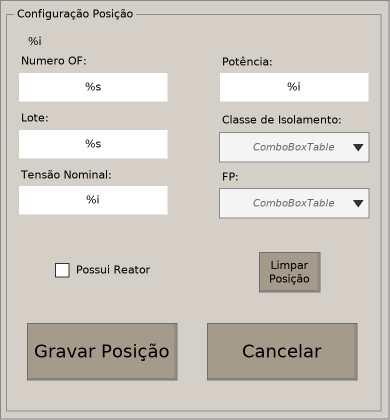
VISUALIZATION ConfigPosicao_2  // 390x420
VAR_IN_OUT
	bReator: BOOL;
	iOFnumber: INT;
	iSrlNumber: INT;
	
	
	
END_VAR
    GroupBox (6,6 375x405), "Configuração Posição"
        Checkbox (47,251 110x26), "Possui Reator", variable: gravarConfigPosicao020.bReator[1]
        Button (21,317 150x57), "Gravar Posição"
            OnMouseClick: CloseDialog Dialog=ConfigPosicao_2, Result=OK, NumpadKeypadSet=True
            OnMouseClick: execute { gravarConfigPosicao020(); }
        Button (201,317 150x57), "Cancelar"
            OnMouseClick: CloseDialog Dialog=ConfigPosicao_2, Result=Cancel, NumpadKeypadSet=True
        Button (253,246 61x40), "Limpar Posição"
            OnMouseClick: CloseDialog Dialog=ConfigPosicao_2, Result=Cancel, NumpadKeypadSet=True
            OnMouseClick: execute {
                gvl_p.aPositionsE020[gvl.actPos].numOF:='0';
                gvl_p.aPositionsE020[gvl.actPos].lote:='0';
                gvl_p.aPositionsE020[gvl.actPos].class:=0;
                gvl_p.aPositionsE020[gvl.actPos].pot:=0;
                gvl_p.aPositionsE020[gvl.actPos].cor:=0;
                IF gvl.totalPos[gvl.actEst] <> 0 THEN
                gvl.totalPos[gvl.actEst]:= gvl.totalPos[gvl.actEst] - 1;
                ELSE
                	gvl.totalPos[gvl.actEst] := 0;
                END_IF
                bReator:=false;
                ///// GERADOR DE LOG -------------------------------------------------------------
                gvl.envialog:= 'Posição Nº ';
                gvl.envialog:= concat(gvl.envialog, INT_TO_STRING(gvl.actPos));
                gvl.envialog:= concat(gvl.envialog,' foi limpa. ESTUFA 020');
                gvl.logRegister20:= gvl.envialog;
            }
        Label (12,40 81x30), "Numero OF:"
    Rectangle (24,30 22x23), "%i", text variable: GVL.actPos
    Textfield (18,72 150x30), "%s", text variable: GVL.cfgPos_OF020
        OnMouseDown: write the text variable via VisuDialogs.Numpad
    Label (18,160 104x30), "Tensão Nominal:"
    Textfield (219,72 150x30), "%i", text variable: GVL.cfgPos_Pot020
        OnMouseDown: write the text variable via VisuDialogs.Numpad
    Label (18,103 81x30), "Lote:"
    Label (219,162 56x30), "FP:"
    Label (219,105 144x30), "Classe de Isolamento:"
    Textfield (18,185 150x30), "%i", text variable: GVL.cfgPos_Class020
        OnMouseDown: write the text variable via VisuDialogs.Numpad
    Label (219,47 56x30), "Potência:"
    Textfield (18,129 150x30), "%s", text variable: GVL.cfgPos_LT020
        OnMouseDown: write the text variable via VisuDialogs.Keypad
    ComboBoxTable (219,132 150x30), variable: GVL.cfgPos_Iso020, data array: GVL_P.arr_Iso_2
        p3854506369: GVL_P.arr_Iso_2[INDEX]
    ComboBoxTable (219,188 150x30), variable: GVL.cfgPos_FP020, data array: GVL_P.arr_FP_2
        p3854506369: GVL_P.arr_FP_2[INDEX]
END_VISUALIZATION

(* stored: Version 1.1.0.1, ProductVersion 3.1.4024.12
   Visu ConfigPosicao_2: Id {f7c709a8-5fe8-4025-b04c-e003caaf7a17} *)
